GLOBALCONSTANTS Computers (* Computers IP Addresses *)
  (* Standard: 61499-1 *)
  (* Version 1.0, 2023-10-22, franz *)
  VAR_GLOBAL CONSTANT
    C_LO : WSTRING := "localhost:61499";
    C_ET : WSTRING := "192.168.5.1:61499"; (* using the IP over USB Virtual Ethernet *)
    C_ST : WSTRING := "192.168.4.1:61499"; (* Using the WIFI Station *)
    C_00 : WSTRING := "192.168.4.1:61499"; (* Using the WIFI Station *)
    C_01 : WSTRING := "192.168.188.1:61499"; (* Student 1 *)
    C_02 : WSTRING := "192.168.188.2:61499"; (* Student 2 *)
    C_03 : WSTRING := "192.168.188.3:61499"; (* Student 3 *)
    C_04 : WSTRING := "192.168.188.4:61499"; (* Student 4 *)
    C_05 : WSTRING := "192.168.188.5:61499"; (* Student 5 *)
    C_06 : WSTRING := "192.168.188.6:61499"; (* Student 6 *)
    C_07 : WSTRING := "192.168.188.7:61499"; (* Student 7 *)
    C_08 : WSTRING := "192.168.188.8:61499"; (* Student 8 *)
    C_09 : WSTRING := "192.168.188.9:61499"; (* Student 9 *)
    C_10 : WSTRING := "192.168.188.10:61499"; (* Student 10 *)
    C_11 : WSTRING := "192.168.188.11:61499"; (* Student 11 *)
    C_12 : WSTRING := "192.168.188.12:61499"; (* Student 12 *)
    C_13 : WSTRING := "192.168.188.13:61499"; (* Student 13 *)
    C_14 : WSTRING := "192.168.188.14:61499"; (* Student 14 *)
    C_15 : WSTRING := "192.168.188.15:61499"; (* Student 15 *)
    C_16 : WSTRING := "192.168.188.16:61499"; (* Student 16 *)
    C_17 : WSTRING := "192.168.188.17:61499"; (* Student 17 *)
    C_18 : WSTRING := "192.168.188.18:61499"; (* Student 18 *)
    C_19 : WSTRING := "192.168.188.19:61499"; (* Student 19 *)
  END_VAR
END_GLOBALCONSTANTS
